VAR_GLOBAL
END_VAR

(* stored: Version 1.1.0.1, ProductVersion 3.1.4024.11
   GVL OP30_Recipe: Id {0a0b9cdf-b491-4b00-891b-67094ea2dee9} *)
